KUKA KRL program: C3_RvR.src

&ACCESS RVO
&PARAM EDITMASK = *
DEFFCT INT C3_RvR( )

   RETURN 1
ENDFCT
